// TIA Portal V17 export
// export: Created 2024-08-26T21:07:17.3244293Z, ExportSetting WithDefaults, DisplayName Totally Integrated Automation Portal, DisplayVersion V17 Update 7, DisplayName TIA Portal Openness, DisplayVersion V17 Update 7, DisplayName TIA Portal Version Control Interface, DisplayVersion V17, DisplayName SINAMICS Startdrive Advanced, DisplayVersion V17 SP2, DisplayName SINAMICS Startdrive G110M, G120, G120C, G120D, G120P, G115D, DisplayVersion V17 SP2, DisplayName SINAMICS Startdrive G130, G150, S120, S150, SINAMICS MV, S210, DisplayVersion V17 SP2, DisplayName STEP 7 Professional, DisplayVersion V17 Update 7, DisplayName STEP 7 Safety, DisplayVersion V17 Update 6, DisplayName WinCC Advanced / Unified PC, DisplayVersion V17 Update 7
DATA_BLOCK "CODE READING NEST"   // DB3
VERSION : 0.1
// stored: AutoNumber true, DBAccessibleFromOPCUA true, DBAccessibleFromWebserver true, InstanceOfName CODE READING, InstanceOfType FB
"CODE READING"
   // VAR_INPUT
   //    hwAdd : HW_IO := 344;
   //    scannerBusy : Bool := FALSE;
   //    autoMode : Bool := FALSE;
   //    manualMode : Bool := TRUE;
   //    scannerReadingComplete : Bool := FALSE;
   //    scannerReadingError : Bool := FALSE;
   //    clearData : Bool := FALSE;
   //    scannerDataSize : Int := 30;
   //    requestScannerAuto : Bool := FALSE;
   //    requestScannerManual : Bool := FALSE;
   //    scannerEnabled : Bool := TRUE;
   //    labelIdentyfier : String[5] := '695';
   //    labelPosition : Int := 13;
   //    labelIdentyfier_2 : String[5] := '';
   //    labelPosition_2 : Int := 0;
   //    label1 : Bool := TRUE;
   //    label2 : Bool := FALSE;
   // END_VAR
   // VAR_OUTPUT
   //    hmiLabel : String[180] := '';
   //    scannerOk : Bool := FALSE;
   //    scannerOk_2 : Bool := FALSE;
   //    clearReadComplete : Bool := FALSE;
   //    requestScannerOutput : Bool := FALSE;
   //    codeRead : Bool := FALSE;
   // END_VAR
   // VAR
   //    scannerReading { ExternalAccessible := 'False'; ExternalVisible := 'False'; ExternalWritable := 'False'} : Array[0..254] of Char;
   //    ScannerReadTimer { S7_SetPoint := 'True'} : TON_TIME;
   // END_VAR
BEGIN
   scannerReading[0] := '$00';
   scannerReading[1] := 'X';
   scannerReading[2] := '$00';
   scannerReading[3] := 'X';
   scannerReading[4] := '$00';
   scannerReading[5] := 'X';
   scannerReading[6] := '$00';
   scannerReading[7] := '$1E';
   scannerReading[8] := 'V';
   scannerReading[9..10] := '0';
   scannerReading[11] := '8';
   scannerReading[12] := '3';
   scannerReading[13] := '4';
   scannerReading[14] := '5';
   scannerReading[15] := 'Y';
   scannerReading[16] := '4';
   scannerReading[17] := '2';
   scannerReading[18] := '5';
   scannerReading[19] := '9';
   scannerReading[20] := '6';
   scannerReading[21] := '9';
   scannerReading[22] := '8';
   scannerReading[23] := 'X';
   scannerReading[24] := 'R';
   scannerReading[25] := '0';
   scannerReading[26..27] := '1';
   scannerReading[28] := '4';
   scannerReading[29] := '6';
   scannerReading[30] := '4';
   scannerReading[31] := '2';
   scannerReading[32] := '4';
   scannerReading[33] := '0';
   scannerReading[34] := '8';
   scannerReading[35] := '0';
   scannerReading[36] := '1';
   scannerReading[37] := '$R';
   scannerReading[38..135] := '$00';
   scannerReading[136..254] := ' ';
   ScannerReadTimer.PT := T#50MS;
   ScannerReadTimer.IN := FALSE;
END_DATA_BLOCK
